Fanuc KAREL source: ka00012.KL

-- PROVISIONAL review KL for V940-1; original PC SHA256 2af565843a017ea9d223c4e57c445cb767c720b2c1f13e1e0c01972dbc9b3799
-- Incomplete behavior may be omitted. Consult companion uncertainty JSON. Do not deploy.
PROGRAM KA00012
%NOLOCKGROUP
VAR
  SRC : INTEGER
-- UNRESOLVED_DECL DST type=002017
BEGIN
  -- V9_ZERO_TABLE_METADATA_HINT layout=0001; no indexed target words; source/name/runtime held
  -- UNRESOLVED_PC offsets 5-16; opcodes 2E,23
  -- UNRESOLVED_PC offsets 21-36; opcodes 21,22,9D,33,B4
  -- UNRESOLVED_PC offsets 41-45; opcodes 7F
END KA00012
